FUNCTION_BLOCK LIMIT_SWITCH_3
  (* Standard: 61499-2 *)
  (* Version 11-01-12, GASR *)
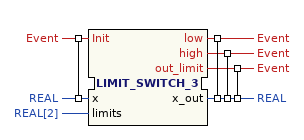
  EVENT_INPUT
    Init WITH x;
  END_EVENT
  EVENT_OUTPUT
    low WITH x_out;
    high WITH x_out;
    out_limit WITH x_out;
  END_EVENT
  VAR_INPUT
    x : REAL;
    limits : ARRAY [0..1] OF REAL := [10,20];
  END_VAR
  VAR_OUTPUT
    x_out : REAL;
  END_VAR
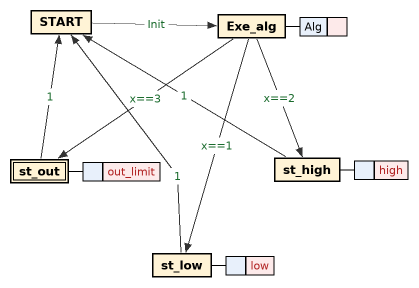
  EC_STATES
    st_out : -> out_limit;
    st_low : -> low;
    START;
    st_high : -> high;
    Exe_alg : Alg;
  END_STATES
  EC_TRANSITIONS
    START TO Exe_alg := Init;
    Exe_alg TO st_out := x==3;
    Exe_alg TO st_low := x==1;
    Exe_alg TO st_high := x==2;
    st_high TO START := 1;
    st_low TO START := 1;
    st_out TO START := 1;
  END_TRANSITIONS
  ALGORITHM Alg IN Lua:
		if limits[1] > x then
			x = 1
		elseif x > limits[2] then
			x = 2
		else
			x = 3
		end
		x_out = x
  END_ALGORITHM
END_FUNCTION_BLOCK
